// Mitsubishi GX Works2 project: z09   PLC: Q02/Q02H

PROGRAM MAIN
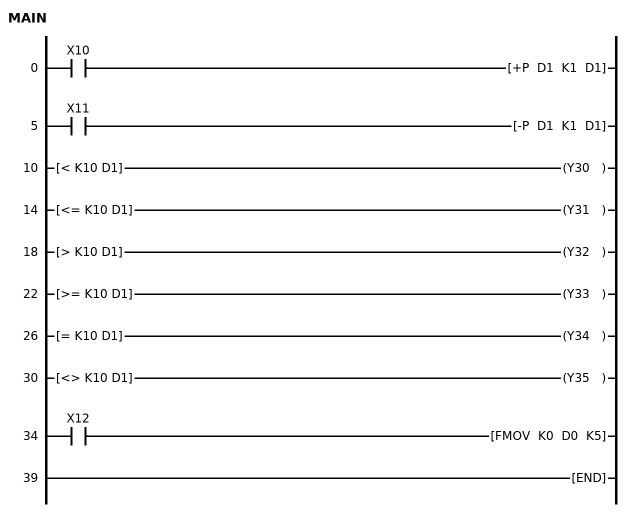
0     LD      X10
      +P      D1 K1 D1
5     LD      X11
      -P      D1 K1 D1
10    LD<     K10 D1
      OUT     Y30
14    LD<=    K10 D1
      OUT     Y31
18    LD>     K10 D1
      OUT     Y32
22    LD>=    K10 D1
      OUT     Y33
26    LD=     K10 D1
      OUT     Y34
30    LD<>    K10 D1
      OUT     Y35
34    LD      X12
      FMOV    K0 D0 K5
39    END
END_PROGRAM
